RoboDK station: Program_VDL_Testobject_AMR_empty.rdk

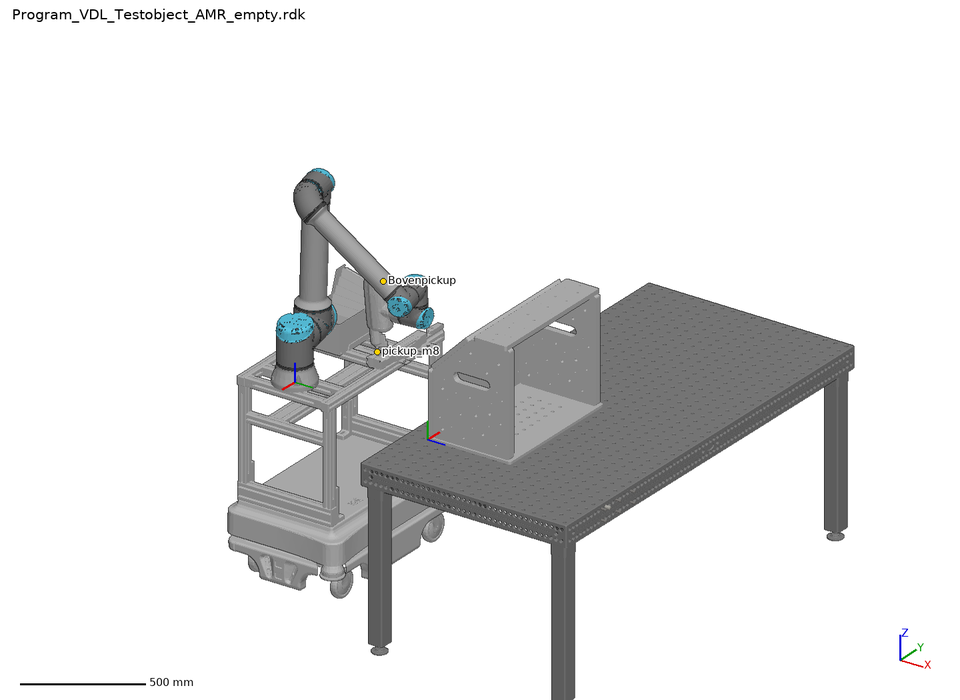
[picture v0: the station drawn from its stored meshes, robots at their saved joint values, targets as dots, program paths as lines]
Station Program_VDL_Testobject_AMR_empty (saved by RoboDK 5.9.6). Poses are relative to the parent item; angles as X-Y-Z fixed-axis rotations.
Station parameters (name, value as stored): CollisionFreePlanner, UR10e, CollisionFreePlanner-Rob UR10e, Simplify-Mesh-Settings
  - object Lastafel at (0, 0, 0) mm, size 1021.8 x 2000 x 842 mm
  - object Lastafel_simplified at (0, 0, 0) mm, size 1000 x 2000 x 802.1 mm
  - frame UR10e Base at (-1574.73, 215.14, 116.62) mm, rotated rx 0 ry 0 rz -90 deg
    - robot UR10e: 6 axes, payload 10 kg, reach 1300 mm, repeatability 0.05 mm, weight 28.9 kg
        modified DH rows (alpha deg, a mm, theta deg, d mm): 0, 0, 0, 180.7; 90, 0, 180, 0; 0, 612.6, 0, 0; 0, 571.335, 0, 174.15; -90, 0, 0, 119.85; 90, 0, 180, 116.55
        joint limits [-300, -150, -30, -360, -360, -360] to [300, 0, 180, 360, 360, 360]; home [30.872, -95.296, 116.362, -22.187, 121.11, 179.827]; saved at [-77.919, -88.358, 129.355, -44.249, -77.326, -92.587]
      - tool schroevendraaier all in met nieuw kopstuk en tool, TCP at (210, -1, 100.6) mm, rotated rx 90 ry -90 rz 90 deg, size 86.2 x 139.7 x 345.9 mm, geometry from schroevendraaier all in met nieuw kopstuk en tool.STEP
      - tool tool simplified, TCP at (210, -1, 100.6) mm, rotated rx 90 ry -90 rz 90 deg, size 86.3 x 139.7 x 346 mm
    - object Assembly mir + frame aangepast naar ur10e versie 2 at (-733.08, 277.19, -552.66) mm, rotated rx 90 ry 0 rz 0.45 deg, size 901.1 x 1139.6 x 580.4 mm, geometry from Assembly mir + frame aangepast naar ur10e versie 2.STEP
    - object Mir + frame simplified at (-733.08, 277.19, -552.66) mm, rotated rx 90 ry 0 rz 0.45 deg, size 925.7 x 1139.7 x 582 mm
  - frame CSV Frame at (-919, 200, 49.99) mm, rotated rx 90 ry 0 rz 90.11 deg
    - object Test object at (0, 0.01, 0) mm, size 650 x 517 x 400 mm, geometry from Test object.STEP
    - object Test object simplified at (0, 0.01, 0) mm, size 650.1 x 517 x 436.5 mm
    - target pickup_m8 (Cartesian target) at (296.95, 143.94, -451.18) mm, rotated rx 9.58 ry 86.75 rz -77.13 deg; joints [-45.747, -65.18, 99.078, -38.37, -45.221, -90.148] of UR10e
    - target Bovenpickup (Cartesian target) at (307.87, 458.95, -429.97) mm, rotated rx -139.66 ry 89.26 rz 129.81 deg; joints [-136.006, -63.802, 89.759, 154.828, 46.597, 89.992] of UR10e
